{attribute 'linkalways'} 
{attribute 'no_explicit_call' := 'This FB is a CLASS and must be accessed using methods or properties'}
{attribute 'enable_dynamic_creation'}
FUNCTION_BLOCK Node_F_VN_MultiplyMatrices EXTENDS VisionNode
VAR
    stSrcMatrix1 : _TcVnMatrix;
    stSrcMatrix2 : _TcVnMatrix;
    stDestMatrix : _TcVnMatrix;
    hrPrev : _HRESULT(S_OK);
	hresult : _HRESULT(S_OK);
END_VAR

METHOD PUBLIC  Clone : I_Node
VAR
	pNode : POINTER TO Node_F_VN_MultiplyMatrices;
END_VAR
pNode := __NEW(Node_F_VN_MultiplyMatrices);
Clone := pNode^;
END_METHOD

METHOD FB_init : BOOL
VAR_INPUT
	bInitRetains : BOOL; // if TRUE, the retain variables are initialized (warm start / cold start)
	bInCopyCode : BOOL;  // if TRUE, the instance afterwards gets moved into the copy code (online change)
END_VAR
AddInput('stSrcMatrix1', stSrcMatrix1);
AddInput('stSrcMatrix2', stSrcMatrix2);
AddInput('hrPrev', hrPrev);
AddOutput('stDestMatrix', stDestMatrix);
AddOutput('hresult',hresult);
END_METHOD

METHOD PROTECTED  OnExecute : HRESULT
hresult.Value := F_VN_MultiplyMatrices(
	stSrcMatrix1 := stSrcMatrix1.Value,
    stSrcMatrix2 := stSrcMatrix2.Value,
    stDestMatrix := stDestMatrix.Value,
	hrPrev:= hrPrev.Value);
END_METHOD

METHOD PUBLIC PreExecutionCheck
VAR_INPUT
	Check : I_PreExecutionChecks;
END_VAR
END_METHOD

END_FUNCTION_BLOCK

(* stored: Version 1.1.0.1, ProductVersion 3.1.4024.13
   POU Node_F_VN_MultiplyMatrices: Id {17f414c9-eaeb-0e1c-3e18-46b86c666e75}, SpecialFunc None
   Folder Constructor: Id {3c11d1f2-6449-0044-2068-abc3e7ba32e2}
   Method Clone: Id {42ef6860-9609-067e-35ca-d2097f49ed1b}
   Method FB_init: Id {51fe7fea-2807-0648-36dc-973fd4ac8700}
   Method OnExecute: Id {dcba4ae7-06d9-0dd7-1ed7-0d0ad3626d9e}
   Method PreExecutionCheck: Id {cee247a7-2dd8-035c-09a6-5f5087cf6c0e} *)
